FUNCTION_BLOCK DrillStation
  (* Standard: 61499-2 *)
  (* Version 0.2, 2003-12-05, JHC, Rockwell Automation, Renamed from NEWCOMPFB. *)
  (* Version 0.1, 2002-01-08, JHC, Rockwell Automation, Added DLY FB as example. *)
  (* Version 0.0, 2000-05-27, JHC, Rockwell Automation *)
  (* Compiler header: package fb.rt.benchmarks.DrillStation; *)
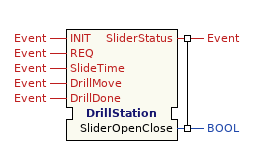
  EVENT_INPUT
    INIT; (* Initialization Request *)
    REQ; (* Normal Execution Request *)
    SlideTime;
    DrillMove;
    DrillDone;
  END_EVENT
  EVENT_OUTPUT
    SliderStatus WITH SliderOpenClose;
  END_EVENT
  VAR_OUTPUT
    SliderOpenClose : BOOL;
  END_VAR
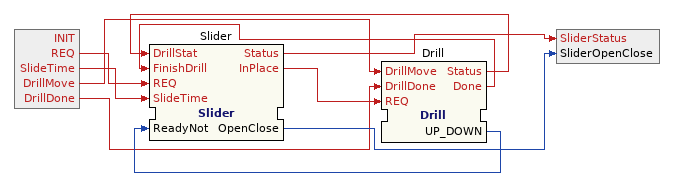
  FBS
    Drill : Drill;
    Slider : Slider;
  END_FBS
  EVENT_CONNECTIONS
    Drill.Status TO Slider.DrillStat;
    Drill.Done TO Slider.FinishDrill;
    REQ TO Slider.REQ;
    SlideTime TO Slider.SlideTime;
    DrillMove TO Drill.DrillMove;
    DrillDone TO Drill.DrillDone;
    Slider.Status TO SliderStatus;
    Slider.InPlace TO Drill.REQ;
  END_CONNECTIONS
  DATA_CONNECTIONS
    Drill.UP_DOWN TO Slider.ReadyNot;
    Slider.OpenClose TO SliderOpenClose;
  END_CONNECTIONS
END_FUNCTION_BLOCK
